(* IEC 61131-3 sources: AXOpen/src/showcase/app/src/components.cognex.vision/Documentation, 12 files *)

(* ---- AxoDataman.st ---- *)
USING AXOpen.Core;

NAMESPACE AXOpen.Components.Cognex.Vision

    {S7.extern=ReadWrite}
    CLASS AxoDataman_Example EXTENDS AXOpen.Core.AxoObject
        //<ComponentDeclaration>
        VAR PUBLIC
            Dataman_280 : AXOpen.Components.Cognex.Vision.v_6_0_0_0.AxoDataman;
        END_VAR
        //</ComponentDeclaration>

        //<InitializationArgumentsDeclaration>
        VAR PUBLIC
            {#ix-set:AttributeName = "<#Activate manual control#>"}
            ActivateManualControl : BOOL;
        END_VAR
        //</InitializationArgumentsDeclaration>

        METHOD PUBLIC OVERRIDE Run
            VAR_INPUT
                inParent : IAxoObject;
            END_VAR

            SUPER.Run(inParent);

            IF ActivateManualControl THEN
                //<DatamanManualControl>
                Dataman_280.ActivateManualControl();
                //</DatamanManualControl>
            END_IF;

            //<Initialization>
            Dataman_280.Run(inParent  :=  THIS, hwID :=  AXOpen.Showcase.HwIdentifiers#cognex_dataman_280_HwID);
            //</Initialization>

            THIS.UseInSequencer();
        END_METHOD

        //<Usage>
        VAR PUBLIC
            Sequencer : AxoSequencer;
            Steps : ARRAY[0..10] OF AXOpen.Core.AxoStep;
        END_VAR

        VAR PRIVATE
            _ResultData  :   AXOpen.Components.Cognex.Vision.v_6_0_0_0.AxoDataman_ResultData;
        END_VAR

        METHOD PRIVATE UseInSequencer
            IF Sequencer.GetContext().OpenCycleCount() <= ULINT#10 THEN
                Sequencer.SequenceMode := eAxoSequenceMode#RunOnce;
            END_IF;

            Sequencer.Run(THIS);
            Sequencer.Open();

            IF(Steps[0].Execute(Sequencer, 'Restore')) THEN
                Dataman_280.Config.InfoTime    := LTIME#2S;
                Dataman_280.Config.ErrorTime   := LTIME#5S;
                Dataman_280.Config.TaskTimeout := LTIME#50S;
                Dataman_280.Restore();
                Sequencer.MoveNext();
            END_IF;

            IF(Steps[1].Execute(Sequencer, 'Clear result data')) THEN
                IF(Dataman_280.ClearResultData().IsDone()) THEN
                    Sequencer.MoveNext();
                END_IF;
            END_IF;

            IF(Steps[2].Execute(Sequencer, 'Read data')) THEN
                IF(Dataman_280.Read().IsDone()) THEN
                    Sequencer.MoveNext();
                END_IF;
            END_IF;

            IF(Steps[3].Execute(Sequencer, 'Evaluate data')) THEN
                _ResultData := Dataman_280.ResultData;
                Sequencer.MoveNext();
            END_IF;

            IF(Steps[4].Execute(Sequencer, 'Restore')) THEN
                Dataman_280.Restore();
                Sequencer.CompleteSequence();
            END_IF;

        END_METHOD

        //</Usage>
    END_CLASS
END_NAMESPACE

(* ---- AxoDataman_Secondary.st ---- *)
USING AXOpen.Core;

NAMESPACE AXOpen.Components.Cognex.Vision

    {S7.extern=ReadWrite}
    CLASS AxoDataman_Secondary_Example EXTENDS AXOpen.Core.AxoObject
        //<ComponentDeclaration>
        VAR PUBLIC
            Dataman_300 : AXOpen.Components.Cognex.Vision.v_6_0_0_0.AxoDataman;
        END_VAR
        //</ComponentDeclaration>

        //<InitializationArgumentsDeclaration>
        VAR PUBLIC
            {#ix-set:AttributeName = "<#Activate manual control#>"}
            ActivateManualControl : BOOL;
        END_VAR
        //</InitializationArgumentsDeclaration>

        METHOD PUBLIC OVERRIDE Run
            VAR_INPUT
                inParent : IAxoObject;
            END_VAR

            SUPER.Run(inParent);

            IF ActivateManualControl THEN
                //<DatamanManualControl>
                Dataman_300.ActivateManualControl();
                //</DatamanManualControl>
            END_IF;

            //<Initialization>
            Dataman_300.Run(inParent := THIS, hwID :=  AXOpen.Showcase.HwIdentifiers#cognex_dataman_380_HwID);
            //</Initialization>

            THIS.UseInSequencer();
        END_METHOD

        //<Usage>
        VAR PUBLIC
            Sequencer : AxoSequencer;
            Steps : ARRAY[0..10] OF AXOpen.Core.AxoStep;
        END_VAR

        VAR PRIVATE
            _ResultData  :   AXOpen.Components.Cognex.Vision.v_6_0_0_0.AxoDataman_ResultData;
        END_VAR

        METHOD PRIVATE UseInSequencer
            IF Sequencer.GetContext().OpenCycleCount() <= ULINT#10 THEN
                Sequencer.SequenceMode := eAxoSequenceMode#RunOnce;
            END_IF;

            Sequencer.Run(THIS);
            Sequencer.Open();

            IF(Steps[0].Execute(Sequencer, 'Restore')) THEN
                Dataman_300.Config.InfoTime    := LTIME#2S;
                Dataman_300.Config.ErrorTime   := LTIME#5S;
                Dataman_300.Config.TaskTimeout := LTIME#50S;
                Dataman_300.Restore();
                Sequencer.MoveNext();
            END_IF;

            IF(Steps[1].Execute(Sequencer, 'Clear result data')) THEN
                IF(Dataman_300.ClearResultData().IsDone()) THEN
                    Sequencer.MoveNext();
                END_IF;
            END_IF;

            IF(Steps[2].Execute(Sequencer, 'Read data')) THEN
                IF(Dataman_300.Read().IsDone()) THEN
                    Sequencer.MoveNext();
                END_IF;
            END_IF;

            IF(Steps[3].Execute(Sequencer, 'Evaluate data')) THEN
                _ResultData := Dataman_300.ResultData;
                Sequencer.MoveNext();
            END_IF;

            IF(Steps[4].Execute(Sequencer, 'Restore')) THEN
                Dataman_300.Restore();
                Sequencer.CompleteSequence();
            END_IF;

        END_METHOD

        //</Usage>
    END_CLASS
END_NAMESPACE

(* ---- AxoDataman_v_6_0_0_0_Showcase.st ---- *)
USING AXOpen.Core;

NAMESPACE AXOpen.Components.Cognex.Vision

    {S7.extern=ReadWrite}
    CLASS AxoDataman_v_6_0_0_0_Showcase EXTENDS AXOpen.Core.AxoObject
        //<ComponentDeclaration>
        VAR PUBLIC
            Dataman_280 : AXOpen.Components.Cognex.Vision.v_6_0_0_0.AxoDataman;
        END_VAR
        //</ComponentDeclaration>

        //<InitializationArgumentsDeclaration>
        VAR PUBLIC
            {#ix-set:AttributeName = "<#Activate manual control#>"}
            ActivateManualControl : BOOL;
        END_VAR
        //</InitializationArgumentsDeclaration>

        METHOD PUBLIC OVERRIDE Run
            VAR_INPUT
                inParent : IAxoObject;
            END_VAR

            SUPER.Run(inParent);

            IF ActivateManualControl THEN
                //<DatamanManualControl>
                Dataman_280.ActivateManualControl();
                //</DatamanManualControl>
            END_IF;

            //<Initialization>
            Dataman_280.Run(inParent  :=  THIS, hwID :=  AXOpen.Showcase.HwIdentifiers#cognex_dataman_280_HwID);
            //</Initialization>

            THIS.UseInSequencer();
        END_METHOD

        //<Usage>
        VAR PUBLIC
            Sequencer : AxoSequencer;
            Steps : ARRAY[0..10] OF AXOpen.Core.AxoStep;
        END_VAR

        VAR PRIVATE
            _ResultData  :   AXOpen.Components.Cognex.Vision.v_6_0_0_0.AxoDataman_ResultData;
        END_VAR

        METHOD PRIVATE UseInSequencer
            IF Sequencer.GetContext().OpenCycleCount() <= ULINT#10 THEN
                Sequencer.SequenceMode := eAxoSequenceMode#RunOnce;
            END_IF;

            Sequencer.Run(THIS);
            Sequencer.Open();

            IF(Steps[0].Execute(Sequencer, 'Restore')) THEN
                Dataman_280.Config.InfoTime    := LTIME#2S;
                Dataman_280.Config.ErrorTime   := LTIME#5S;
                Dataman_280.Config.TaskTimeout := LTIME#50S;
                Dataman_280.Restore();
                Sequencer.MoveNext();
            END_IF;

            IF(Steps[1].Execute(Sequencer, 'Clear result data')) THEN
                IF(Dataman_280.ClearResultData().IsDone()) THEN
                    Sequencer.MoveNext();
                END_IF;
            END_IF;

            IF(Steps[2].Execute(Sequencer, 'Read data')) THEN
                IF(Dataman_280.Read().IsDone()) THEN
                    Sequencer.MoveNext();
                END_IF;
            END_IF;

            IF(Steps[3].Execute(Sequencer, 'Evaluate data')) THEN
                _ResultData := Dataman_280.ResultData;
                Sequencer.MoveNext();
            END_IF;

            IF(Steps[4].Execute(Sequencer, 'Restore')) THEN
                Dataman_280.Restore();
                Sequencer.CompleteSequence();
            END_IF;

        END_METHOD

        //</Usage>
    END_CLASS
END_NAMESPACE

(* ---- AxoDataman_v_6_0_0_0_Showcase2.st ---- *)
USING AXOpen.Core;

NAMESPACE AXOpen.Components.Cognex.Vision

    {S7.extern=ReadWrite}
    CLASS AxoDataman_v_6_0_0_0_Showcase2 EXTENDS AXOpen.Core.AxoObject
        //<ComponentDeclaration>
        VAR PUBLIC
            Dataman_300 : AXOpen.Components.Cognex.Vision.v_6_0_0_0.AxoDataman;
        END_VAR
        //</ComponentDeclaration>

        //<InitializationArgumentsDeclaration>
        VAR PUBLIC
            {#ix-set:AttributeName = "<#Activate manual control#>"}
            ActivateManualControl : BOOL;
        END_VAR
        //</InitializationArgumentsDeclaration>

        METHOD PUBLIC OVERRIDE Run
            VAR_INPUT
                inParent : IAxoObject;
            END_VAR

            SUPER.Run(inParent);

            IF ActivateManualControl THEN
                //<DatamanManualControl>
                Dataman_300.ActivateManualControl();
                //</DatamanManualControl>
            END_IF;

            //<Initialization>
            Dataman_300.Run(inParent := THIS, hwID :=  AXOpen.Showcase.HwIdentifiers#cognex_dataman_380_HwID);
            //</Initialization>

            THIS.UseInSequencer();
        END_METHOD

        //<Usage>
        VAR PUBLIC
            Sequencer : AxoSequencer;
            Steps : ARRAY[0..10] OF AXOpen.Core.AxoStep;
        END_VAR

        VAR PRIVATE
            _ResultData  :   AXOpen.Components.Cognex.Vision.v_6_0_0_0.AxoDataman_ResultData;
        END_VAR

        METHOD PRIVATE UseInSequencer
            IF Sequencer.GetContext().OpenCycleCount() <= ULINT#10 THEN
                Sequencer.SequenceMode := eAxoSequenceMode#RunOnce;
            END_IF;

            Sequencer.Run(THIS);
            Sequencer.Open();

            IF(Steps[0].Execute(Sequencer, 'Restore')) THEN
                Dataman_300.Restore();
                Sequencer.MoveNext();
            END_IF;

            IF(Steps[1].Execute(Sequencer, 'Clear result data')) THEN
                IF(Dataman_300.ClearResultData().IsDone()) THEN
                    Sequencer.MoveNext();
                END_IF;
            END_IF;

            IF(Steps[2].Execute(Sequencer, 'Read data')) THEN
                IF(Dataman_300.Read().IsDone()) THEN
                    Sequencer.MoveNext();
                END_IF;
            END_IF;

            IF(Steps[3].Execute(Sequencer, 'Evaluate data')) THEN
                _ResultData := Dataman_300.ResultData;
                Sequencer.MoveNext();
            END_IF;

            IF(Steps[4].Execute(Sequencer, 'Restore')) THEN
                Dataman_300.Restore();
                Sequencer.CompleteSequence();
            END_IF;

        END_METHOD

        //</Usage>
    END_CLASS
END_NAMESPACE

(* ---- AxoInsight_v_24_0_0.st ---- *)
USING AXOpen.Core;

NAMESPACE AXOpen.Components.Cognex.Vision

    {S7.extern=ReadWrite}
    CLASS AxoInsight_v_24_0_0_Example EXTENDS AXOpen.Core.AxoObject
        //<ComponentDeclaration>
        VAR PUBLIC
            Insight_2800 : AXOpen.Components.Cognex.Vision.v_24_0_0.AxoInsight;
        END_VAR
        //</ComponentDeclaration>

        //<InitializationArgumentsDeclaration>
        VAR PUBLIC
            {#ix-set:AttributeName = "<#Activate manual control#>"}
            ActivateManualControl : BOOL;
        END_VAR
        //</InitializationArgumentsDeclaration>

        METHOD PUBLIC OVERRIDE Run
            VAR_INPUT
                inParent : IAxoObject;
            END_VAR

            SUPER.Run(inParent);

            IF ActivateManualControl THEN
                //<InsightManualControl>
                Insight_2800.ActivateManualControl();
                //</InsightManualControl>
            END_IF;

            //<Initialization>
            Insight_2800.Run(inParent := THIS, hwID := AXOpen.Showcase.HwIdentifiers#cognex_insight_2800_HwID);
            //</Initialization>
            THIS.UseInSequencer();
        END_METHOD

        //<Usage>
        VAR PUBLIC
            Sequencer : AxoSequencer;
            Steps : ARRAY[0..14] OF AXOpen.Core.AxoStep;
        END_VAR

        VAR PRIVATE
            _InspectionResults  :   AXOpen.Components.Cognex.Vision.v_24_0_0.AxoInsight_ResultData;
            _UserData           :   AXOpen.Components.Cognex.Vision.v_24_0_0.AxoInsight_UserData;
        END_VAR

        METHOD PRIVATE UseInSequencer
            IF Sequencer.GetContext().OpenCycleCount() <= ULINT#10 THEN
                Sequencer.SequenceMode := eAxoSequenceMode#RunOnce;
            END_IF;

            Sequencer.Run(THIS);
            Sequencer.Open();

            IF(Steps[0].Execute(Sequencer, 'Restore')) THEN
                Insight_2800.Config.InfoTime    := LTIME#10S;
                Insight_2800.Config.ErrorTime   := LTIME#50S;
                Insight_2800.Config.TaskTimeout := LTIME#50S;
                Insight_2800.Restore();
                Sequencer.MoveNext();
            END_IF;

            IF(Steps[1].Execute(Sequencer, 'Change job by number:2')) THEN
                IF(Insight_2800.ChangeJob(UINT#2).IsDone()) THEN
                    Sequencer.MoveNext();
                END_IF;
            END_IF;

            IF(Steps[2].Execute(Sequencer, 'Change job by name:1_BOGE_Lavy_pedal_090_091')) THEN
                IF(Insight_2800.ChangeJob('1_BOGE_Lavy_pedal_090_091').IsDone()) THEN
                    Sequencer.MoveNext();
                END_IF;
            END_IF;

            IF(Steps[3].Execute(Sequencer, 'Trigger')) THEN
                IF(Insight_2800.Trigger().IsDone()) THEN
                    Sequencer.MoveNext();
                END_IF;
            END_IF;

            IF(Steps[4].Execute(Sequencer, 'Evaluate inspection results')) THEN
                _InspectionResults := Insight_2800.InspectionResults;
                Sequencer.MoveNext();
            END_IF;

            IF(Steps[5].Execute(Sequencer, 'Clear inspection results')) THEN
                IF(Insight_2800.ClearInspectionResults().IsDone()) THEN
                    Sequencer.MoveNext();
                END_IF;
            END_IF;

            IF(Steps[6].Execute(Sequencer, 'Soft event:5')) THEN
                IF(Insight_2800.SoftEvent(UINT#5).IsDone()) THEN
                    Sequencer.MoveNext();
                END_IF;
            END_IF;

            IF(Steps[7].Execute(Sequencer, 'Clear user data')) THEN
                IF(Insight_2800.ClearUserData().IsDone()) THEN
                    Sequencer.MoveNext();
                END_IF;
            END_IF;

            IF(Steps[8].Execute(Sequencer, 'Set user data as byte')) THEN
                IF(Insight_2800.SetUserDataAsByte(BYTE#12,UINT#0)) THEN
                    Sequencer.MoveNext();
                END_IF;
            END_IF;

            IF(Steps[9].Execute(Sequencer, 'Set user data as string')) THEN
                IF(Insight_2800.SetUserDataAsString('Set user data string l24',UINT#1)) THEN
                    Sequencer.MoveNext();
                END_IF;
            END_IF;

            IF(Steps[10].Execute(Sequencer, 'Set user data as dint')) THEN
                IF(Insight_2800.SetUserDataAsDint(DINT#123456,UINT#25)) THEN
                    Sequencer.MoveNext();
                END_IF;
            END_IF;

            IF(Steps[11].Execute(Sequencer, 'Set user data as real')) THEN
                IF(Insight_2800.SetUserDataAsReal(REAL#789.123,UINT#29)) THEN
                    Sequencer.MoveNext();
                END_IF;
            END_IF;

            IF(Steps[12].Execute(Sequencer, 'Send already prepared user data')) THEN
                IF(Insight_2800.SendUserData().IsDone()) THEN
                    Sequencer.MoveNext();
                END_IF;
            END_IF;

            IF(Steps[13].Execute(Sequencer, 'Send user data passed as input variable')) THEN
                _UserData.Data[0] := BYTE#65;
                // ..
                // ..
                _UserData.Data[27] := BYTE#32;

                IF(Insight_2800.SendUserData(_UserData, UINT#32).IsDone()) THEN
                    Sequencer.MoveNext();
                END_IF;
            END_IF;

            IF(Steps[14].Execute(Sequencer, 'Restore')) THEN
                Insight_2800.Restore();
                Sequencer.CompleteSequence();
            END_IF;
        END_METHOD

        //</Usage>

    END_CLASS
END_NAMESPACE

(* ---- AxoInsight_v_24_0_0_Showcase.st ---- *)
USING AXOpen.Core;

NAMESPACE AXOpen.Components.Cognex.Vision

    {S7.extern=ReadWrite}
    CLASS AxoInsight_v_24_0_0_Showcase EXTENDS AXOpen.Core.AxoObject
        //<ComponentDeclaration>
        VAR PUBLIC
            Insight_2800 : AXOpen.Components.Cognex.Vision.v_24_0_0.AxoInsight;
        END_VAR
        //</ComponentDeclaration>

        //<InitializationArgumentsDeclaration>
        VAR PUBLIC
            {#ix-set:AttributeName = "<#Activate manual control#>"}
            ActivateManualControl : BOOL;
        END_VAR
        //</InitializationArgumentsDeclaration>

        METHOD PUBLIC OVERRIDE Run
            VAR_INPUT
                inParent : IAxoObject;
            END_VAR

            SUPER.Run(inParent);

            IF ActivateManualControl THEN
                //<InsightManualControl>
                Insight_2800.ActivateManualControl();
                //</InsightManualControl>
            END_IF;

            //<Initialization>
            Insight_2800.Run(inParent := THIS, hwID := AXOpen.Showcase.HwIdentifiers#cognex_insight_2800_HwID);
            //</Initialization>
            THIS.UseInSequencer();
        END_METHOD

        //<Usage>
        VAR PUBLIC
            Sequencer : AxoSequencer;
            Steps : ARRAY[0..14] OF AXOpen.Core.AxoStep;
        END_VAR

        VAR PRIVATE
            _InspectionResults  :   AXOpen.Components.Cognex.Vision.v_24_0_0.AxoInsight_ResultData;
            _UserData           :   AXOpen.Components.Cognex.Vision.v_24_0_0.AxoInsight_UserData;
        END_VAR

        METHOD PRIVATE UseInSequencer
            IF Sequencer.GetContext().OpenCycleCount() <= ULINT#10 THEN
                Sequencer.SequenceMode := eAxoSequenceMode#RunOnce;
            END_IF;

            Sequencer.Run(THIS);
            Sequencer.Open();

            IF(Steps[0].Execute(Sequencer, 'Restore')) THEN
                Insight_2800.Restore();
                Sequencer.MoveNext();
            END_IF;

            IF(Steps[1].Execute(Sequencer, 'Change job by number:2')) THEN
                IF(Insight_2800.ChangeJob(UINT#2).IsDone()) THEN
                    Sequencer.MoveNext();
                END_IF;
            END_IF;

            IF(Steps[2].Execute(Sequencer, 'Change job by name:1_BOGE_Lavy_pedal_090_091')) THEN
                IF(Insight_2800.ChangeJob('1_BOGE_Lavy_pedal_090_091').IsDone()) THEN
                    Sequencer.MoveNext();
                END_IF;
            END_IF;

            IF(Steps[3].Execute(Sequencer, 'Trigger')) THEN
                IF(Insight_2800.Trigger().IsDone()) THEN
                    Sequencer.MoveNext();
                END_IF;
            END_IF;

            IF(Steps[4].Execute(Sequencer, 'Evaluate inspection results')) THEN
                _InspectionResults := Insight_2800.InspectionResults;
                Sequencer.MoveNext();
            END_IF;

            IF(Steps[5].Execute(Sequencer, 'Clear inspection results')) THEN
                IF(Insight_2800.ClearInspectionResults().IsDone()) THEN
                    Sequencer.MoveNext();
                END_IF;
            END_IF;

            IF(Steps[6].Execute(Sequencer, 'Soft event:5')) THEN
                IF(Insight_2800.SoftEvent(UINT#5).IsDone()) THEN
                    Sequencer.MoveNext();
                END_IF;
            END_IF;

            IF(Steps[7].Execute(Sequencer, 'Clear user data')) THEN
                IF(Insight_2800.ClearUserData().IsDone()) THEN
                    Sequencer.MoveNext();
                END_IF;
            END_IF;

            IF(Steps[8].Execute(Sequencer, 'Set user data as byte')) THEN
                IF(Insight_2800.SetUserDataAsByte(BYTE#12,UINT#0)) THEN
                    Sequencer.MoveNext();
                END_IF;
            END_IF;

            IF(Steps[9].Execute(Sequencer, 'Set user data as string')) THEN
                IF(Insight_2800.SetUserDataAsString('Set user data string l24',UINT#1)) THEN
                    Sequencer.MoveNext();
                END_IF;
            END_IF;

            IF(Steps[10].Execute(Sequencer, 'Set user data as dint')) THEN
                IF(Insight_2800.SetUserDataAsDint(DINT#123456,UINT#25)) THEN
                    Sequencer.MoveNext();
                END_IF;
            END_IF;

            IF(Steps[11].Execute(Sequencer, 'Set user data as real')) THEN
                IF(Insight_2800.SetUserDataAsReal(REAL#789.123,UINT#29)) THEN
                    Sequencer.MoveNext();
                END_IF;
            END_IF;

            IF(Steps[12].Execute(Sequencer, 'Send already prepared user data')) THEN
                IF(Insight_2800.SendUserData().IsDone()) THEN
                    Sequencer.MoveNext();
                END_IF;
            END_IF;

            IF(Steps[13].Execute(Sequencer, 'Send user data passed as input variable')) THEN
                _UserData.Data[0] := BYTE#65;
                // ..
                // ..
                _UserData.Data[27] := BYTE#32;

                IF(Insight_2800.SendUserData(_UserData, UINT#32).IsDone()) THEN
                    Sequencer.MoveNext();
                END_IF;
            END_IF;

            IF(Steps[14].Execute(Sequencer, 'Restore')) THEN
                Insight_2800.Restore();
                Sequencer.CompleteSequence();
            END_IF;
        END_METHOD

        //</Usage>

    END_CLASS
END_NAMESPACE

(* ---- AxoInsight_v_6_0_0.st ---- *)
USING AXOpen.Core;

NAMESPACE AXOpen.Components.Cognex.Vision

    {S7.extern=ReadWrite}
    CLASS AxoInsight_v_6_0_0_Example EXTENDS AXOpen.Core.AxoObject
        //<ComponentDeclaration>
        VAR PUBLIC
            Insight_7600 : AXOpen.Components.Cognex.Vision.v_6_0_0_0.AxoInsight;
        END_VAR
        //</ComponentDeclaration>

        //<InitializationArgumentsDeclaration>
        VAR PUBLIC
            {#ix-set:AttributeName = "<#Activate manual control#>"}
            ActivateManualControl : BOOL;
        END_VAR
        //</InitializationArgumentsDeclaration>

        METHOD PUBLIC OVERRIDE Run
            VAR_INPUT
                inParent : IAxoObject;
            END_VAR

            SUPER.Run(inParent);

            IF ActivateManualControl THEN
                //<InsightManualControl>
                Insight_7600.ActivateManualControl();
                //</InsightManualControl>
            END_IF;

            //<Initialization>
            Insight_7600.Run(inParent := THIS, hwID :=  AXOpen.Showcase.HwIdentifiers#cognex_insight_7600_HwID);
            //</Initialization>
            THIS.UseInSequencer();
        END_METHOD

        //<Usage>
        VAR PUBLIC
            Sequencer : AxoSequencer;
            Steps : ARRAY[0..14] OF AXOpen.Core.AxoStep;
        END_VAR

        VAR PRIVATE
            _InspectionResults  :   AXOpen.Components.Cognex.Vision.v_6_0_0_0.AxoInsight_ResultData;
            _UserData           :   AXOpen.Components.Cognex.Vision.v_6_0_0_0.AxoInsight_UserData;
        END_VAR

        METHOD PRIVATE UseInSequencer
            IF Sequencer.GetContext().OpenCycleCount() <= ULINT#10 THEN
                Sequencer.SequenceMode := eAxoSequenceMode#RunOnce;
            END_IF;

            Sequencer.Run(THIS);
            Sequencer.Open();

            IF(Steps[0].Execute(Sequencer, 'Restore')) THEN
                Insight_7600.Config.InfoTime    := LTIME#10S;
                Insight_7600.Config.ErrorTime   := LTIME#50S;
                Insight_7600.Config.TaskTimeout := LTIME#50S;
                Insight_7600.Restore();
                Sequencer.MoveNext();
            END_IF;

            IF(Steps[1].Execute(Sequencer, 'Change job by number:2')) THEN
                IF(Insight_7600.ChangeJob(UINT#2).IsDone()) THEN
                    Sequencer.MoveNext();
                END_IF;
            END_IF;

            IF(Steps[2].Execute(Sequencer, 'Change job: 1_test01.job')) THEN
                IF(Insight_7600.ChangeJob('1_test01.job').IsDone()) THEN
                    Sequencer.MoveNext();
                END_IF;
            END_IF;

            IF(Steps[3].Execute(Sequencer, 'Trigger')) THEN
                IF(Insight_7600.Trigger().IsDone()) THEN
                    Sequencer.MoveNext();
                END_IF;
            END_IF;

            IF(Steps[4].Execute(Sequencer, 'Evaluate inspection results')) THEN
                _InspectionResults := Insight_7600.InspectionResults;
                Sequencer.MoveNext();
            END_IF;

            IF(Steps[5].Execute(Sequencer, 'Clear inspaction results')) THEN
                IF(Insight_7600.ClearInspectionResults().IsDone()) THEN
                    Sequencer.MoveNext();
                END_IF;
            END_IF;

            IF(Steps[6].Execute(Sequencer, 'Soft event:5')) THEN
                IF(Insight_7600.SoftEvent(UINT#5).IsDone()) THEN
                    Sequencer.MoveNext();
                END_IF;
            END_IF;

            IF(Steps[7].Execute(Sequencer, 'Clear user data')) THEN
                IF(Insight_7600.ClearUserData().IsDone()) THEN
                    Sequencer.MoveNext();
                END_IF;
            END_IF;

            IF(Steps[8].Execute(Sequencer, 'Set user data as byte')) THEN
                IF(Insight_7600.SetUserDataAsByte(BYTE#12,UINT#0)) THEN
                    Sequencer.MoveNext();
                END_IF;
            END_IF;

            IF(Steps[9].Execute(Sequencer, 'Set user data as string')) THEN
                IF(Insight_7600.SetUserDataAsString('Set user data string l24',UINT#1)) THEN
                    Sequencer.MoveNext();
                END_IF;
            END_IF;

            IF(Steps[10].Execute(Sequencer, 'Set user data as dint')) THEN
                IF(Insight_7600.SetUserDataAsDint(DINT#123456,UINT#25)) THEN
                    Sequencer.MoveNext();
                END_IF;
            END_IF;

            IF(Steps[11].Execute(Sequencer, 'Set user data as real')) THEN
                IF(Insight_7600.SetUserDataAsReal(REAL#789.123,UINT#29)) THEN
                    Sequencer.MoveNext();
                END_IF;
            END_IF;

            IF(Steps[12].Execute(Sequencer, 'Send already prepared user data')) THEN
                IF(Insight_7600.SendUserData().IsDone()) THEN
                    Sequencer.MoveNext();
                END_IF;
            END_IF;

            IF(Steps[13].Execute(Sequencer, 'Send user data passed as input variable')) THEN
                _UserData.Data[0] := BYTE#65;
                // ..
                // ..
                _UserData.Data[27] := BYTE#32;

                IF(Insight_7600.SendUserData(_UserData, UINT#32).IsDone()) THEN
                    Sequencer.MoveNext();
                END_IF;
            END_IF;

            IF(Steps[14].Execute(Sequencer, 'Restore')) THEN
                Insight_7600.Restore();
                Sequencer.CompleteSequence();
            END_IF;
        END_METHOD

        //</Usage>

    END_CLASS
END_NAMESPACE

(* ---- AxoInsight_v_6_0_0_0_Showcase.st ---- *)
USING AXOpen.Core;

NAMESPACE AXOpen.Components.Cognex.Vision

    {S7.extern=ReadWrite}
    CLASS AxoInsight_v_6_0_0_0_Showcase EXTENDS AXOpen.Core.AxoObject
        //<ComponentDeclaration>
        VAR PUBLIC
            Insight_7600 : AXOpen.Components.Cognex.Vision.v_6_0_0_0.AxoInsight;
        END_VAR
        //</ComponentDeclaration>

        //<InitializationArgumentsDeclaration>
        VAR PUBLIC
            {#ix-set:AttributeName = "<#Activate manual control#>"}
            ActivateManualControl : BOOL;
        END_VAR
        //</InitializationArgumentsDeclaration>

        METHOD PUBLIC OVERRIDE Run
            VAR_INPUT
                inParent : IAxoObject;
            END_VAR

            SUPER.Run(inParent);

            IF ActivateManualControl THEN
                //<InsightManualControl>
                Insight_7600.ActivateManualControl();
                //</InsightManualControl>
            END_IF;

            //<Initialization>
            Insight_7600.Run(inParent := THIS, hwID :=  AXOpen.Showcase.HwIdentifiers#cognex_insight_7600_HwID);
            //</Initialization>
            THIS.UseInSequencer();
        END_METHOD

        //<Usage>
        VAR PUBLIC
            Sequencer : AxoSequencer;
            Steps : ARRAY[0..14] OF AXOpen.Core.AxoStep;
        END_VAR

        VAR PRIVATE
            _InspectionResults  :   AXOpen.Components.Cognex.Vision.v_6_0_0_0.AxoInsight_ResultData;
            _UserData           :   AXOpen.Components.Cognex.Vision.v_6_0_0_0.AxoInsight_UserData;
        END_VAR

        METHOD PRIVATE UseInSequencer
            IF Sequencer.GetContext().OpenCycleCount() <= ULINT#10 THEN
                Sequencer.SequenceMode := eAxoSequenceMode#RunOnce;
            END_IF;

            Sequencer.Run(THIS);
            Sequencer.Open();

            IF(Steps[0].Execute(Sequencer, 'Restore')) THEN
                Insight_7600.Config.InfoTime    := LTIME#10S;
                Insight_7600.Config.ErrorTime   := LTIME#50S;
                Insight_7600.Config.TaskTimeout := LTIME#50S;
                Insight_7600.Restore();
                Sequencer.MoveNext();
            END_IF;

            IF(Steps[1].Execute(Sequencer, 'Change job by number:2')) THEN
                IF(Insight_7600.ChangeJob(UINT#2).IsDone()) THEN
                    Sequencer.MoveNext();
                END_IF;
            END_IF;

            IF(Steps[2].Execute(Sequencer, 'Change job: 1_test01.job')) THEN
                IF(Insight_7600.ChangeJob('1_test01.job').IsDone()) THEN
                    Sequencer.MoveNext();
                END_IF;
            END_IF;

            IF(Steps[3].Execute(Sequencer, 'Trigger')) THEN
                IF(Insight_7600.Trigger().IsDone()) THEN
                    Sequencer.MoveNext();
                END_IF;
            END_IF;

            IF(Steps[4].Execute(Sequencer, 'Evaluate inspection results')) THEN
                _InspectionResults := Insight_7600.InspectionResults;
                Sequencer.MoveNext();
            END_IF;

            IF(Steps[5].Execute(Sequencer, 'Clear inspaction results')) THEN
                IF(Insight_7600.ClearInspectionResults().IsDone()) THEN
                    Sequencer.MoveNext();
                END_IF;
            END_IF;

            IF(Steps[6].Execute(Sequencer, 'Soft event:5')) THEN
                IF(Insight_7600.SoftEvent(UINT#5).IsDone()) THEN
                    Sequencer.MoveNext();
                END_IF;
            END_IF;

            IF(Steps[7].Execute(Sequencer, 'Clear user data')) THEN
                IF(Insight_7600.ClearUserData().IsDone()) THEN
                    Sequencer.MoveNext();
                END_IF;
            END_IF;

            IF(Steps[8].Execute(Sequencer, 'Set user data as byte')) THEN
                IF(Insight_7600.SetUserDataAsByte(BYTE#12,UINT#0)) THEN
                    Sequencer.MoveNext();
                END_IF;
            END_IF;

            IF(Steps[9].Execute(Sequencer, 'Set user data as string')) THEN
                IF(Insight_7600.SetUserDataAsString('Set user data string l24',UINT#1)) THEN
                    Sequencer.MoveNext();
                END_IF;
            END_IF;

            IF(Steps[10].Execute(Sequencer, 'Set user data as dint')) THEN
                IF(Insight_7600.SetUserDataAsDint(DINT#123456,UINT#25)) THEN
                    Sequencer.MoveNext();
                END_IF;
            END_IF;

            IF(Steps[11].Execute(Sequencer, 'Set user data as real')) THEN
                IF(Insight_7600.SetUserDataAsReal(REAL#789.123,UINT#29)) THEN
                    Sequencer.MoveNext();
                END_IF;
            END_IF;

            IF(Steps[12].Execute(Sequencer, 'Send already prepared user data')) THEN
                IF(Insight_7600.SendUserData().IsDone()) THEN
                    Sequencer.MoveNext();
                END_IF;
            END_IF;

            IF(Steps[13].Execute(Sequencer, 'Send user data passed as input variable')) THEN
                _UserData.Data[0] := BYTE#65;
                // ..
                // ..
                _UserData.Data[27] := BYTE#32;

                IF(Insight_7600.SendUserData(_UserData, UINT#32).IsDone()) THEN
                    Sequencer.MoveNext();
                END_IF;
            END_IF;

            IF(Steps[14].Execute(Sequencer, 'Restore')) THEN
                Insight_7600.Restore();
                Sequencer.CompleteSequence();
            END_IF;
        END_METHOD

        //</Usage>

    END_CLASS
END_NAMESPACE

(* ---- AxoVisionPro.st ---- *)
USING AXOpen.Core;

NAMESPACE AXOpen.Components.Cognex.Vision

    {S7.extern=ReadWrite}
    CLASS AxoVisionPro_Example EXTENDS AXOpen.Core.AxoObject
        //<ComponentDeclaration>
        VAR PUBLIC
            VisionPro : AXOpen.Components.Cognex.Vision.AxoVisionPro;
        END_VAR
        //</ComponentDeclaration>

        //<InitializationArgumentsDeclaration>
        VAR PUBLIC
            {#ix-set:AttributeName = "<#Activate manual control#>"}
            ActivateManualControl : BOOL;
        END_VAR
        //</InitializationArgumentsDeclaration>

        METHOD PUBLIC OVERRIDE Run
            VAR_INPUT
                inParent : IAxoObject;
            END_VAR

            SUPER.Run(inParent);

            IF ActivateManualControl THEN
                //<InsightManualControl>
                VisionPro.ActivateManualControl();
                //</InsightManualControl>
            END_IF;

            //<Initialization>
            VisionPro.Run(inParent := THIS, hwID := AXOpen.Showcase.HwIdentifiers#vision_pro_HwID, CameraNo := BYTE#1);
            //</Initialization>
            THIS.UseInSequencer();
        END_METHOD

        //<Usage>
        VAR PUBLIC
            Sequencer : AxoSequencer;
            Steps : ARRAY[0..10] OF AXOpen.Core.AxoStep;
        END_VAR

        VAR PRIVATE
            _InspectionResults : ARRAY[0..1300] OF BYTE;
            _UserData : ARRAY[0..1300] OF BYTE;
        END_VAR

        METHOD PRIVATE UseInSequencer
            IF Sequencer.GetContext().OpenCycleCount() <= ULINT#10 THEN
                Sequencer.SequenceMode := eAxoSequenceMode#RunOnce;
            END_IF;

            Sequencer.Run(THIS);
            Sequencer.Open();

            IF(Steps[0].Execute(Sequencer, 'Restore')) THEN
                VisionPro.Config.InfoTime    := LTIME#5S;
                VisionPro.Config.ErrorTime   := LTIME#10S;
                VisionPro.Config.TaskTimeout := LTIME#50S;
                VisionPro.Restore();
                Sequencer.MoveNext();
            END_IF;

            IF(Steps[1].Execute(Sequencer, 'HardResetAllCameras')) THEN
                IF(VisionPro.HardResetAllCameras().IsDone()) THEN
                    Sequencer.MoveNext();
                END_IF;
            END_IF;

            IF(Steps[2].Execute(Sequencer, 'SendData')) THEN
                IF(VisionPro.SendData(InspectionType := BYTE#1, BufferID := BYTE#0, JobID := BYTE#1, Length := UINT#1, Data := _UserData).IsDone()) THEN
                    Sequencer.MoveNext();
                END_IF;
            END_IF;

            IF(Steps[3].Execute(Sequencer, 'Trigger')) THEN
                IF(VisionPro.Trigger().IsDone()) THEN
                    Sequencer.MoveNext();
                END_IF;
            END_IF;

            IF(Steps[4].Execute(Sequencer, 'SendData')) THEN
                IF(VisionPro.SendData(InspectionType := BYTE#2, BufferID := BYTE#0, JobID := BYTE#1, Length := UINT#1, Data := _UserData).IsDone()) THEN
                    Sequencer.MoveNext();
                END_IF;
            END_IF;

            IF(Steps[5].Execute(Sequencer, 'ReadResults')) THEN
                IF(VisionPro.ReadResults(JobID := BYTE#1, Length := UINT#620, Data := _InspectionResults).IsDone()) THEN
                    Sequencer.MoveNext();
                END_IF;
            END_IF;

            IF(Steps[6].Execute(Sequencer, 'Reset')) THEN
                IF(VisionPro.Reset().IsDone()) THEN
                    Sequencer.MoveNext();
                END_IF;
            END_IF;

            IF(Steps[7].Execute(Sequencer, 'Restore')) THEN
                VisionPro.Restore();
                Sequencer.CompleteSequence();
            END_IF;
        END_METHOD

        //</Usage>

    END_CLASS
END_NAMESPACE

(* ---- AxoVisionPro_Showcase.st ---- *)
USING AXOpen.Core;

NAMESPACE AXOpen.Components.Cognex.Vision

    {S7.extern=ReadWrite}
    CLASS AxoVisionPro_Showcase EXTENDS AXOpen.Core.AxoObject
        //<ComponentDeclaration>
        VAR PUBLIC
            VisionPro : AXOpen.Components.Cognex.Vision.AxoVisionPro;
        END_VAR
        //</ComponentDeclaration>

        //<InitializationArgumentsDeclaration>
        VAR PUBLIC
            {#ix-set:AttributeName = "<#Activate manual control#>"}
            ActivateManualControl : BOOL;
        END_VAR
        //</InitializationArgumentsDeclaration>

        METHOD PUBLIC OVERRIDE Run
            VAR_INPUT
                inParent : IAxoObject;
            END_VAR

            SUPER.Run(inParent);

            IF ActivateManualControl THEN
                //<InsightManualControl>
                VisionPro.ActivateManualControl();
                //</InsightManualControl>
            END_IF;

            //<Initialization>
            VisionPro.Run(inParent := THIS, hwID := AXOpen.Showcase.HwIdentifiers#vision_pro_HwID, CameraNo := BYTE#1);
            //</Initialization>
            THIS.UseInSequencer();
        END_METHOD

        //<Usage>
        VAR PUBLIC
            Sequencer : AxoSequencer;
            Steps : ARRAY[0..10] OF AXOpen.Core.AxoStep;
        END_VAR

        VAR PRIVATE
            _InspectionResults : ARRAY[0..1300] OF BYTE;
            _UserData : ARRAY[0..1300] OF BYTE;
        END_VAR

        METHOD PRIVATE UseInSequencer
            IF Sequencer.GetContext().OpenCycleCount() <= ULINT#10 THEN
                Sequencer.SequenceMode := eAxoSequenceMode#RunOnce;
            END_IF;

            Sequencer.Run(THIS);
            Sequencer.Open();

            IF(Steps[0].Execute(Sequencer, 'Restore')) THEN
                VisionPro.Restore();
                Sequencer.MoveNext();
            END_IF;

            IF(Steps[1].Execute(Sequencer, 'HardResetAllCameras')) THEN
                IF(VisionPro.HardResetAllCameras().IsDone()) THEN
                    Sequencer.MoveNext();
                END_IF;
            END_IF;

            IF(Steps[2].Execute(Sequencer, 'SendData')) THEN
                IF(VisionPro.SendData(InspectionType := BYTE#1, BufferID := BYTE#0, JobID := BYTE#1, Length := UINT#1, Data := _UserData).IsDone()) THEN
                    Sequencer.MoveNext();
                END_IF;
            END_IF;

            IF(Steps[3].Execute(Sequencer, 'Trigger')) THEN
                IF(VisionPro.Trigger().IsDone()) THEN
                    Sequencer.MoveNext();
                END_IF;
            END_IF;

            IF(Steps[4].Execute(Sequencer, 'SendData')) THEN
                IF(VisionPro.SendData(InspectionType := BYTE#2, BufferID := BYTE#0, JobID := BYTE#1, Length := UINT#1, Data := _UserData).IsDone()) THEN
                    Sequencer.MoveNext();
                END_IF;
            END_IF;

            IF(Steps[5].Execute(Sequencer, 'ReadResults')) THEN
                IF(VisionPro.ReadResults(JobID := BYTE#1, Length := UINT#620, Data := _InspectionResults).IsDone()) THEN
                    Sequencer.MoveNext();
                END_IF;
            END_IF;

            IF(Steps[6].Execute(Sequencer, 'Reset')) THEN
                IF(VisionPro.Reset().IsDone()) THEN
                    Sequencer.MoveNext();
                END_IF;
            END_IF;

            IF(Steps[7].Execute(Sequencer, 'Restore')) THEN
                VisionPro.Restore();
                Sequencer.CompleteSequence();
            END_IF;
        END_METHOD

        //</Usage>

    END_CLASS
END_NAMESPACE

(* ---- AxoVisionProNet.st ---- *)
USING AXOpen.Core;

NAMESPACE AXOpen.Components.Cognex.Vision

    {S7.extern=ReadWrite}
    CLASS AxoVisionProNet_Example EXTENDS AXOpen.Core.AxoObject
        //<ComponentDeclaration>
        VAR PUBLIC
            VisionProNet : AXOpen.Components.Cognex.Vision.AxoVisionProNet;
        END_VAR
        //</ComponentDeclaration>

        //<InitializationArgumentsDeclaration>
        VAR PUBLIC
            {#ix-set:AttributeName = "<#Activate manual control#>"}
            ActivateManualControl : BOOL;
        END_VAR
        //</InitializationArgumentsDeclaration>

        METHOD PUBLIC OVERRIDE Run
            VAR_INPUT
                inParent : IAxoObject;
            END_VAR

            SUPER.Run(inParent);

            IF ActivateManualControl THEN
                //<VisionProNetManualControl>
                VisionProNet.ActivateManualControl();
                //</VisionProNetManualControl>
            END_IF;

            //<Initialization>
            // AxoVisionProNet talks to the Vision PC over TCP via its .NET twin.
            // The socket is opened from Program.cs (InitializeVisionClientAsync);
            // here we only configure timeouts and run the component cyclically.
            VisionProNet.Config.InfoTime    := LTIME#5S;
            VisionProNet.Config.ErrorTime   := LTIME#10S;
            VisionProNet.Config.TaskTimeout := LTIME#50S;
            VisionProNet.Run(inParent := THIS);
            //</Initialization>

            THIS.UseInSequencer();
        END_METHOD

        //<Usage>
        VAR PUBLIC
            Sequencer : AxoSequencer;
            Steps : ARRAY[0..10] OF AXOpen.Core.AxoStep;
        END_VAR

        METHOD PRIVATE UseInSequencer
            IF Sequencer.GetContext().OpenCycleCount() <= ULINT#10 THEN
                Sequencer.SequenceMode := eAxoSequenceMode#RunOnce;
            END_IF;

            Sequencer.Run(THIS);
            Sequencer.Open();

            // Restore clears all remote tasks and seeds the recipe / part
            // identification carried in every Vision PC request.
            IF(Steps[0].Execute(Sequencer, 'Restore and set part identification')) THEN
                VisionProNet.Control.VariantId := 'VARIANT-A';
                VisionProNet.Control.PartId    := 'PART-0001';
                VisionProNet.Control.TriggerId := INT#1;
                VisionProNet.Restore();
                Sequencer.MoveNext();
            END_IF;

            // Select the inspection recipe / job on the Vision PC.
            IF(Steps[1].Execute(Sequencer, 'Select recipe on Vision PC')) THEN
                IF(VisionProNet.SetRecipe().IsDone()) THEN
                    Sequencer.MoveNext();
                END_IF;
            END_IF;

            // Fire an inspection for the configured TriggerId / PartId.
            IF(Steps[2].Execute(Sequencer, 'Trigger inspection')) THEN
                IF(VisionProNet.Trigger().IsDone()) THEN
                    Sequencer.MoveNext();
                END_IF;
            END_IF;

            // Pull the inspection verdict back from the Vision PC.
            IF(Steps[3].Execute(Sequencer, 'Read inspection result')) THEN
                IF(VisionProNet.InspectionResult().IsDone()) THEN
                    Sequencer.MoveNext();
                END_IF;
            END_IF;

            // Combined path: send application-specific payload AND trigger in one
            // gated task (disabled by the component while Trigger/SetRecipe run).
            IF(Steps[4].Execute(Sequencer, 'Trigger with specific data')) THEN
                IF(VisionProNet.TriggerWithSpecificData().IsDone()) THEN
                    Sequencer.MoveNext();
                END_IF;
            END_IF;

            // Receive the typed result payload into the specific-data container.
            IF(Steps[5].Execute(Sequencer, 'Receive specific data')) THEN
                IF(VisionProNet.ReceiveSpecificData().IsDone()) THEN
                    Sequencer.MoveNext();
                END_IF;
            END_IF;

            // Error recovery: a remote task that faulted (e.g. Vision PC offline,
            // request rejected) raises HasRemoteException. Restore() clears every
            // task back to idle so the sequence can be re-run.
            IF(Steps[6].Execute(Sequencer, 'Error recovery')) THEN
                //<VisionProNetErrorRecovery>
                IF VisionProNet.TriggerTask.HasRemoteException
                    OR VisionProNet.SetRecipeTask.HasRemoteException
                    OR VisionProNet.InspectionResultTask.HasRemoteException
                    OR VisionProNet.TriggerWithSpecificDataTask.HasRemoteException
                    OR VisionProNet.ReceiveSpecificDataTask.HasRemoteException THEN
                    VisionProNet.Restore();
                END_IF;
                //</VisionProNetErrorRecovery>
                Sequencer.CompleteSequence();
            END_IF;
        END_METHOD
        //</Usage>

        // Commissioning-only task. The component gates SendSpecificDataAndTypes on
        // manual mode, so it is invoked from a manual-control helper rather than the
        // automatic sequence. Activate manual control (ActivateManualControl) first.
        METHOD PUBLIC CommissioningSendData : IAxoTaskState
            //<VisionProNetCommissioning>
            CommissioningSendData := VisionProNet.SendSpecificDataAndTypes();
            //</VisionProNetCommissioning>
        END_METHOD

    END_CLASS
END_NAMESPACE

(* ---- CognexVision.st ---- *)
USING AXOpen.Components.Cognex.Vision;

NAMESPACE AXOpen.Components.Cognex.Vision

    {S7.extern=ReadWrite}
    CLASS CognexVision EXTENDS AXOpen.Core.AxoObject
        VAR PUBLIC
            _rootObject :   AxoObject;
            axoInsight_v_6_0_0_0 : AxoInsight_v_6_0_0_Example;
            axoDataman_v_6_0_0_0 : AxoDataman_Example;
            axoDataman_v_6_0_0_0_2 : AxoDataman_Secondary_Example;
            axoInsight_v_24_0_0 : AxoInsight_v_24_0_0_Example;
            axoVisionPro : AxoVisionPro_Example;
        END_VAR

        METHOD PUBLIC Execute
            _rootObject.Run(THIS);
            axoInsight_v_6_0_0_0.Run(_rootObject);
            axoDataman_v_6_0_0_0.Run(_rootObject);
            axoDataman_v_6_0_0_0_2.Run(_rootObject);
            axoInsight_v_24_0_0.Run(_rootObject);
            axoVisionPro.Run(_rootObject);
        END_METHOD
    END_CLASS
END_NAMESPACE
